# EPICS autosave request: iocs/asiTpxIOC/iocBoot/iocASItpx/auto_settings.req
file "asiTpx_settings.req",       P=$(P),  R=cam1:
file "NDStdArrays_settings.req",  P=$(P),  R=image1:
file "commonPlugin_settings.req", P=$(P)
